// TIA Portal V16 export
// export: Created 2023-03-29T11:05:03.064957Z, ExportSetting WithDefaults, DisplayName Totally Integrated Automation Portal, DisplayVersion V16 Update 6, DisplayName TIA Portal Version Control Interface, DisplayVersion V16 Update 2, DisplayName TIA Portal Openness, DisplayVersion V16 Update 6, DisplayName STEP 7 Professional, DisplayVersion V16 Update 6, DisplayName STEP 7 Safety, DisplayVersion V16, DisplayName WinCC Advanced, DisplayVersion V16 Update 6
DATA_BLOCK "Alarm-Pompownia-Sucho-Max_DB"   // DB143
AUTHOR : rtecmer
VERSION : 0.1
// stored: AutoNumber true, DBAccessibleFromOPCUA true, InstanceOfName Alarm-Pompownia-Sucho-Max, InstanceOfType FB
"Alarm-Pompownia-Sucho-Max"
   // VAR_OUTPUT
   //    bit_on_alarm_bar_max_pompownia { ExternalWritable := 'False'} : Bool;
   // END_VAR
   // VAR
   //    bit_max_pompownia { ExternalAccessible := 'False'; ExternalVisible := 'False'; ExternalWritable := 'False'} : Bool;
   //    bit_normalne_pompownia { ExternalAccessible := 'False'; ExternalVisible := 'False'; ExternalWritable := 'False'} : Bool;
   //    "bit_max _bar_B7" { ExternalAccessible := 'False'; ExternalVisible := 'False'; ExternalWritable := 'False'} : Bool;
   //    bit_off_alarm_max_pompownia { ExternalAccessible := 'False'; ExternalVisible := 'False'; ExternalWritable := 'False'} : Bool;
   // END_VAR
BEGIN
END_DATA_BLOCK
